// SIMATIC S7-200 project (STEP 7-Micro/WIN), CPU 224 REL 02.01

SYMBOL_TABLE USER1
DI21_4           V4.4
DI21_3           V3.4
DI21_2           V2.4
DI21_1           V1.4
chlodzenie       VW140
grzanie          VW130
tz               VW120
t                VW100
histereza        VW110
PT100            AIW8
Cooling          Q0.0
Heating          Q0.2
IDLE             Q0.1
T_gora           I0.1
T_dol            I0.2
H_gora           I0.4
H_dol            I0.5
END_SYMBOL_TABLE

ORGANIZATION_BLOCK MAIN:OB1
TITLE=
BEGIN
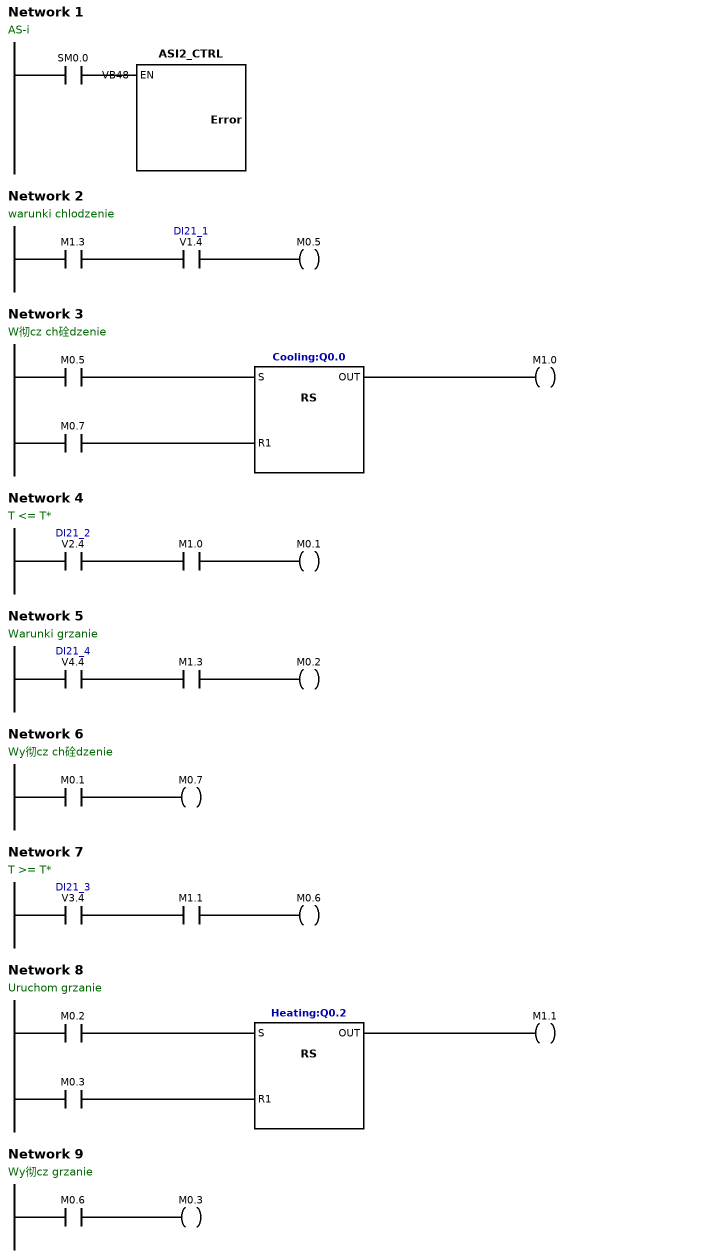
Network 1
// AS-i
// (network saved uncompiled; LAD cells follow)
// row 0: c0 -| |- SM0.0  c1 [ASI2_CTRL Error EN:=VB48]
// row 1: c1 [box]
Network 2
// warunki chlodzenie
LD     M1.3
A      DI21_1:V1.4
=      M0.5
Network 3
// W彻cz ch硂dzenie
// (network saved uncompiled; LAD cells follow)
// row 0: c0 -| |- M0.5  c1 --  c2 [RS Cooling:Q0.0 S:=power@row0, R1:=power@row1, OUT=>power]  c3 --  c4 -( ) M1.0
// row 1: c0 -| |- M0.7  c1 --  c2 [box]
Network 4
// T <= T*
LD     DI21_2:V2.4
A      M1.0
=      M0.1
Network 5
// Warunki grzanie
LD     DI21_4:V4.4
A      M1.3
=      M0.2
Network 6
// Wy彻cz ch硂dzenie
LD     M0.1
=      M0.7
Network 7
// T >= T*
LD     DI21_3:V3.4
A      M1.1
=      M0.6
Network 8
// Uruchom grzanie
// (network saved uncompiled; LAD cells follow)
// row 0: c0 -| |- M0.2  c1 --  c2 [RS Heating:Q0.2 S:=power@row0, R1:=power@row1, OUT=>power]  c3 --  c4 -( ) M1.1
// row 1: c0 -| |- M0.3  c1 --  c2 [box]
Network 9
// Wy彻cz grzanie
LD     M0.6
=      M0.3
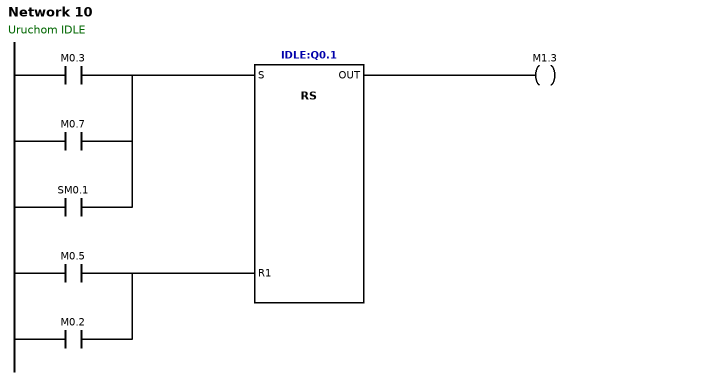
Network 10
// Uruchom IDLE
// (network saved uncompiled; LAD cells follow)
// row 0: c0 -| |- M0.3 v  c1 --  c2 [RS IDLE:Q0.1 S:=power@row0, R1:=power@row3, OUT=>power]  c3 --  c4 -( ) M1.3
// row 1: c0 -| |- M0.7 ^v  c2 [box]
// row 2: c0 -| |- SM0.1 ^  c2 [box]
// row 3: c0 -| |- M0.5 v  c1 --  c2 [box]
// row 4: c0 -| |- M0.2 ^
END_ORGANIZATION_BLOCK

// SBR1: protected block, not included

// SBR2: protected block, not included

// SBR3: protected block, not included
